RoboDK station: Robot7_2TCP.rdk

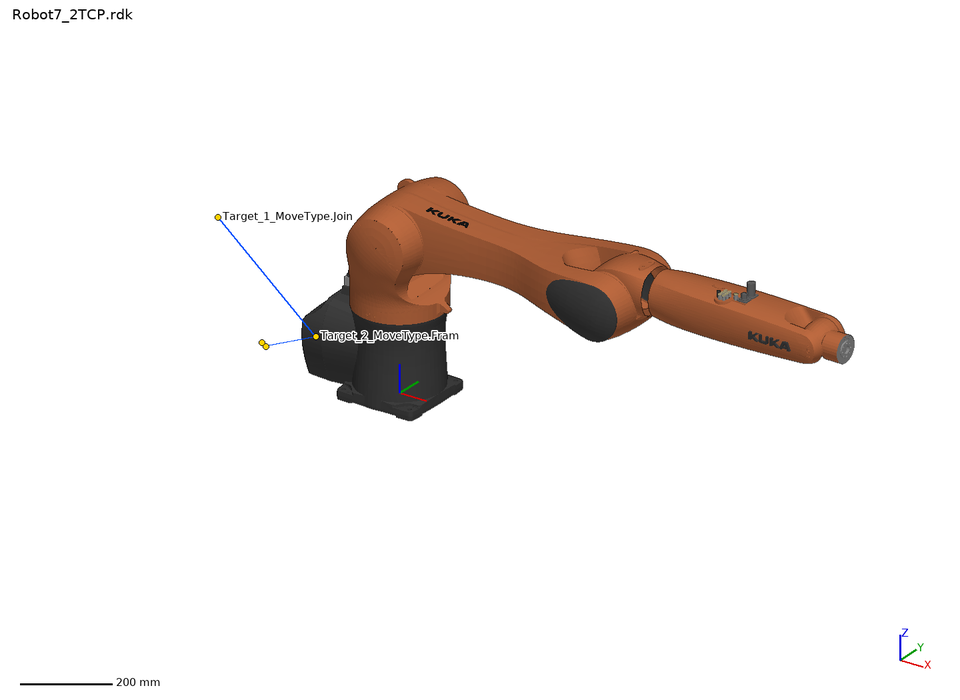
[picture v0: the station drawn from its stored meshes, robots at their saved joint values, targets as dots, program paths as lines]
Station Robot7_2TCP. Poses are relative to the parent item; angles as X-Y-Z fixed-axis rotations.
  - frame Base at (0, 0, 0) mm
    - robot Linear Axis: 1 axes
        modified DH rows (alpha deg, a mm, theta deg, d mm): 0, 0, 0, 0 linear
        base shift (0, 0, 0) mm, rotated rx 0 ry 90 rz 0 deg
        joint limits [-1000] to [1000]; home [0]; saved at [0]
      - robot Robot (model KUKA KR 10 R1100 sixx): 6 axes, payload 10 kg, reach 1101 mm, repeatability 0.03 mm, weight 54 kg
          modified DH rows (alpha deg, a mm, theta deg, d mm): 0, 0, 0, 400; -90, 25, 0, 0; 0, 560, -90, 0; -90, 35, 0, 515; 90, 0, 0, 0; -90, 0, 180, 80
          joint limits [-170, -190, -120, -185, -120, -350] to [170, 45, 156, 185, 120, 350]; home [0, -90, 90, 0, 0, 0]; saved at [0, 0, 0, 0, 0, 0]
        - tool Greifer1, TCP at (43.5, -78.7, 129.7) mm, rotated rx 90 ry 0 rz 0 deg
        - tool Greifer2, TCP at (40, 0, 186.7) mm
    - target Target_1_MoveType.Joint (joint target) at (13.37, -704.56, 708.97) mm, rotated rx -8.36 ry 61.57 rz -178.7 deg; joints [84.043, -57.261, 115.707, 78.815, -83.207, 59.112, 0] of Robot
    - target Target_2_MoveType.Frame (Cartesian target) at (267.8, -697.9, 489.2) mm, rotated rx 0 ry 0 rz -97.11 deg; joints [89.428, -53.485, 115.756, 83.195, -86.436, 62.483, 58.82] of Robot
    - target Target_3_MoveType.Frame (Cartesian target) at (267.8, -886.68, 541.6) mm, rotated rx -45 ry 0 rz 180 deg; joints [69.706, -62.509, 96.967, 49.728, 18.75, 27.165, 58.82] of Robot
    - target Target_4_MoveType.Frame (Cartesian target) at (267.8, -900.82, 555.75) mm, rotated rx -45 ry 0 rz 180 deg; joints [70.085, -62.04, 94.422, 44.972, 19.925, 32.427, 58.82] of Robot
  - program Prg (16 instructions, listed below)
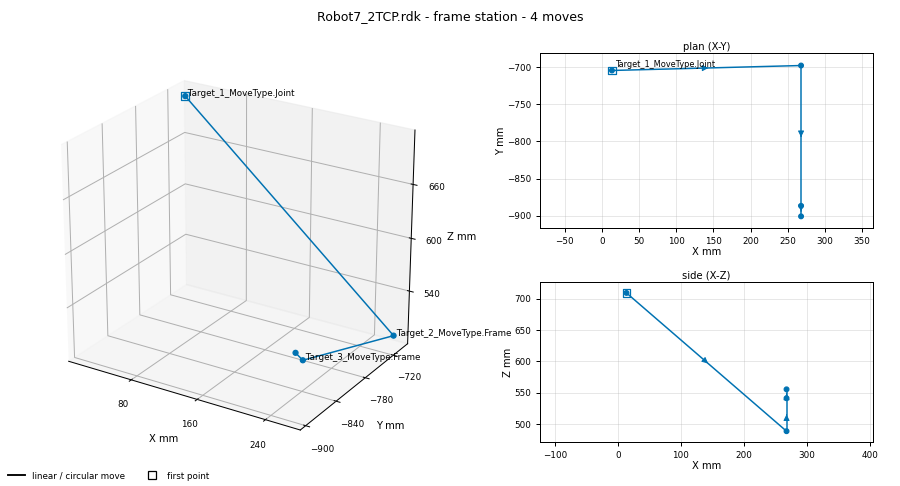
[picture p0: tool path of Robot7_2TCP.rdk in frame station, 4 of 4 moves have a stored position in this frame; points joined in program order, loops and branches not executed]

--- program Prg (robot Robot) ---
  Set Tool: Greifer1
  Smooth(10)
  Set speed (225.0 deg/s)
  MoveJ (Target_1_MoveType.Joint)
  Set Tool: Greifer1
  Smooth(10)
  Set speed (2000.0 mm/s)
  MoveL (Target_2_MoveType.Frame)
  Set Tool: Greifer1
  Smooth(10)
  Set speed (2000.0 mm/s)
  MoveL (Target_3_MoveType.Frame)
  Set Tool: Greifer1
  Smooth(0)
  Set speed (2000.0 mm/s)
  MoveL (Target_4_MoveType.Frame)
